FUNCTION_BLOCK EtherCATFactory
VAR
	DynamicMemoryManager : FB_DynMem_Manager2;
END_VAR

END_FUNCTION_BLOCK

(* stored: Version 1.1.0.1, ProductVersion 3.1.4024.12
   POU EtherCATFactory: Id {068d6bf7-c72d-464f-947f-295d84e58383}, SpecialFunc None *)
